PROGRAM MAIN
VAR
	xInsertion : Insertion;
	
	xServoNC : LinearServoNC;
	xClearLinkMC : LinearClearLinkMC;
	xAirPiston : LinearAirPiston;
	xSimplePiston : SimplePiston;
END_VAR

(*
this solution contains the package for various motion devices and the inheritance hierarchy, and any additional types
the Insertion Package folder under DUTs + WithinTolerance() can be copied to any project/module as needed

I_Drive contains the minimum behavior for any drive
FBA_Drive implements I_Drive with the minimum declaration
	FBA_TrifectaDrive extends it by adding an outer limit sensor for drives requiring 3 sensors
	
all Insertion-capable drives extend FBA_Drive or FBA_TrifectaDrive and implement I_ContinuousDrive, I_PositionalDrive, or I_EncodedDrive
*)

END_PROGRAM

(* stored: Version 1.1.0.1, ProductVersion 3.1.4024.11
   POU MAIN: Id {fd6b2cef-77a7-4c3e-b06c-08694f2c3803}, SpecialFunc None *)
